// TIA Portal V20 export
FUNCTION "TrapezoidalProfile_Linear_Cal" : Void   // FC61, SCL
// stored: Access Published, SetENOAutomatically false
   VAR_INPUT
      CPM : LReal;
      travelDistance : LReal;
   END_VAR
   VAR_OUTPUT
      distance : LReal;
      velocity : LReal;
      acceleration : LReal;
      deceleration : LReal;
      jerk : LReal;
   END_VAR
   VAR_TEMP
      CycleTime : LReal;
   END_VAR
   VAR CONSTANT
      PI : LReal := 3.14159265;
   END_VAR
BEGIN
   REGION Velocity
       #CycleTime := (60.0 / #CPM) / 2.0;
       #distance := #travelDistance;
       #velocity := 1.5 * #travelDistance / #CycleTime;
       #acceleration := 4.5 * #travelDistance / (#CycleTime * #CycleTime);
       #deceleration := #acceleration;
       #jerk := 0.0;
   END_REGION
END_FUNCTION
